FUNCTION IsValidContainer : BOOL
VAR_INPUT
    Container : ITcVnContainer;
END_VAR

IsValidContainer := Container <> 0;

END_FUNCTION

(* stored: Version 1.1.0.1, ProductVersion 3.1.4024.13
   POU IsValidContainer: Id {28bdfab1-acc8-4d33-8d0a-eabac17c8d76}, SpecialFunc None *)
